TYPE ST_TcpVisionParCmd :
STRUCT
    Reserved : BOOL;
END_STRUCT
END_TYPE

(* stored: Version 1.1.0.1, ProductVersion 3.1.4024.12
   DUT ST_TcpVisionParCmd: Id {0c1dc300-b198-43a4-888f-d7d9af6b979a} *)
